(* PLC project StorageFixture, greenforge-labs codescribe-fixture 1 *)
(* stored: creationDateTime 2020-01-01T00:00:00 *)

PROGRAM FBD_STORAGE
  VAR
    tmr : TON;
    pulse : TP;
  END_VAR

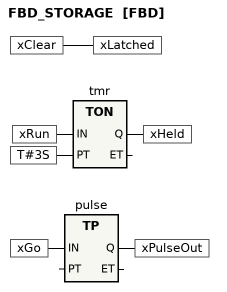
(* FBD diagram, written out as Structured Text *)
IF xClear THEN xLatched := FALSE; END_IF;
tmr(IN := xRun, PT := T#3S, Q => xHeld);
pulse(IN := xGo, Q => xPulseOut);
END_PROGRAM
